// TIA Portal V17 export
// export: Created 2023-03-08T16:44:23.1874801Z, ExportSetting None, DisplayName Totally Integrated Automation Portal, DisplayVersion V17 Update 4, DisplayName TIA Portal Openness, DisplayVersion V17 Update 4, DisplayName TIA Portal Version Control Interface, DisplayVersion V17, DisplayName STEP 7 Professional, DisplayVersion V17 Update 4, DisplayName STEP 7 Safety, DisplayVersion V17, DisplayName WinCC Advanced / Unified PC, DisplayVersion V17 Update 4
DATA_BLOCK "DI"   // DB12
{ S7_Optimized_Access := 'TRUE' }
// stored: AutoNumber false, MemoryReserve 100
   VAR
      DI1 : Bool;   // DIGITAL INPUT 1
      DI2 : Bool;   // DIGITAL INPUT 2
      DI3 : Bool;   // DIGITAL INPUT 3
      DI4 : Bool;   // DIGITAL INPUT 4
      DI5 : Bool;   // DIGITAL INPUT 5
      DI6 : Bool;   // DIGITAL INPUT 6
      DI7 : Bool;   // DIGITAL INPUT 7
      DI8 : Bool;   // DIGITAL INPUT 8
      DI9 : Bool;   // DIGITAL INPUT 9
      DI10 : Bool;   // DIGITAL INPUT 10
      DI11 : Bool;   // DIGITAL INPUT 11
      DI12 : Bool;   // DIGITAL INPUT 12
      DI13 : Bool;   // DIGITAL INPUT 13
      DI14 : Bool;   // DIGITAL INPUT 14
      DI15 : Bool;   // DIGITAL INPUT 15
      DI16 : Bool;   // DIGITAL INPUT 16
      DI17 : Bool;   // DIGITAL INPUT 17
      DI18 : Bool;   // DIGITAL INPUT 18
      DI19 : Bool;   // DIGITAL INPUT 19
      DI20 : Bool;   // DIGITAL INPUT 20
      DA1 : Bool;   // DIGITAL ALARM 1
      DA2 : Bool;   // DIGITAL ALARM 2
      DA3 : Bool;   // DIGITAL ALARM 3
      DA4 : Bool;   // DIGITAL ALARM 4
   END_VAR
BEGIN
END_DATA_BLOCK
